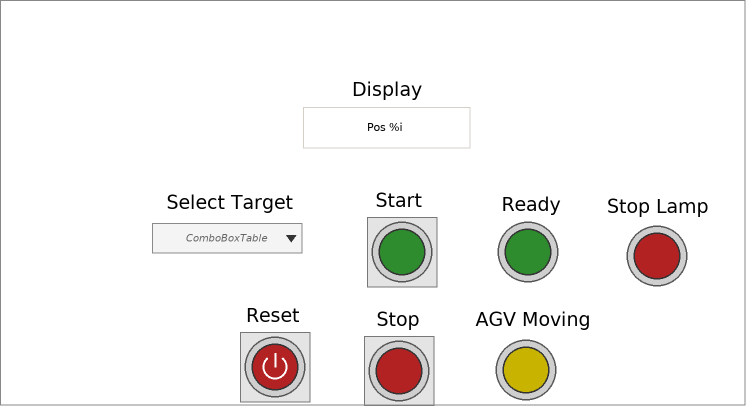
VISUALIZATION HMIoperator  // 746x406, background image Display.Display
    PowerSwitch (240,332 70x70), variable: GVL.qxResetButton, input disabled if: NOT SFC.ResetMemory, behaviour: TOGGLE, style: Switch-PowerSwitch-Red
    PushSwitchLed (367,217 70x70), variable: GVL.qxStartButton, input disabled if: GVL.ixAGVMoving, behaviour: TOGGLE, style: Switch-PushSwitchLed-Green
    PushSwitchLed (364,336 70x70), variable: GVL.qxStopButton, input disabled if: NOT GVL.ixAGVMoving, behaviour: TOGGLE, style: Switch-PushSwitchLed-Red
    ComboBoxTable (152,223 150x30), variable: SFC.TargIndex, input disabled if: GVL.ixAGVMoving, data array: SFC.Target
        p3854506369: SFC.Target[INDEX]
    Lamp1 (493,217 70x70), variable: SFC.qxGreenLamp, style: Lamp-Lamp1-Green
    Textfield (303,107 167x41), "Pos %i", text variable: GVL.iiAtPos, invisible if: GVL.ixAGVMoving
    Rectangle (142,189 176x27), "Select Target"
    Rectangle (570,193 176x27), "Stop Lamp"
    Rectangle (445,306 176x27), "AGV Moving"
    Lamp1 (491,335 70x70), variable: SFC.MovingLamp, style: Lamp-Lamp1-Yellow
    Rectangle (352,186 94x29), "Start"
    Rectangle (351,305 94x29), "Stop"
    Rectangle (226,301 94x29), "Reset"
    Rectangle (299,76 176x27), "Display"
    Lamp1 (622,221 70x70), variable: SFC.qxRedLamp, style: Lamp-Lamp1-Red
    Rectangle (443,191 176x27), "Ready"
END_VISUALIZATION

(* stored: Version 1.1.0.1, ProductVersion 3.1.4024.12
   Visu HMIoperator: Id {3f59e3be-c288-499f-95b0-32b5b3b63ab0} *)
